PROGRAM MAIN
VAR
	fbScaling : FB_Scaling;
END_VAR

P_ControlBox(); // Run selected control box mode (virtual or real)
fbScaling();

END_PROGRAM

(* stored: Version 1.1.0.1, ProductVersion 3.1.4024.12
   POU MAIN: Id {34467066-1969-4a23-bd22-a8eb1fd5af96}, SpecialFunc None *)
